// TIA Portal V20 export
FUNCTION_BLOCK "Side_Hydraulic"   // FB4, LAD
{ S7_Optimized_Access := 'TRUE' }
// stored: MemoryReserve 100, SetENOAutomatically false
   VAR_INPUT
      setUp : Bool;
      setDown : Bool;
      manual_Up : Bool;
      manual_Down : Bool;
      Sensor1_Up : Bool;
      Sensor1_Down : Bool;
      Sensor2_Up : Bool;
      Sensor2_Down : Bool;
      Reset : Bool;
   END_VAR
   VAR_OUTPUT
      Actuator_Up : Bool;
      Actuator_Down : Bool;
      Hydraulic_Unit : Bool;
      Alarm_Push_Actuators : Bool;
      Alarm_Pull_Actuators : Bool;
      Sensors_Down : Bool;
      Sensors_Up : Bool;
      Error : Bool;
   END_VAR
   VAR
      Time_to_PUSH_actuator { ExternalAccessible := 'False'; ExternalVisible := 'False'; ExternalWritable := 'False'} : TON_TIME;
      Time_to_PULL_actuator { S7_SetPoint := 'True'} : TON_TIME;
      Hydraulic_Unit_Timer { S7_SetPoint := 'True'} : TOF_TIME;
      TIMER_Pallet_UP { S7_SetPoint := 'True'} : TOF_TIME;
      TIMER_Pallet_DOWN { S7_SetPoint := 'True'} : TOF_TIME;
      Timer_Error { S7_SetPoint := 'True'} : TON_TIME;
      command_UP { ExternalAccessible := 'False'; ExternalVisible := 'False'; ExternalWritable := 'False'} : Bool;
      command_Down { ExternalAccessible := 'False'; ExternalVisible := 'False'; ExternalWritable := 'False'} : Bool;
   END_VAR
BEGIN

REGION Network 1: Sensors DOWN
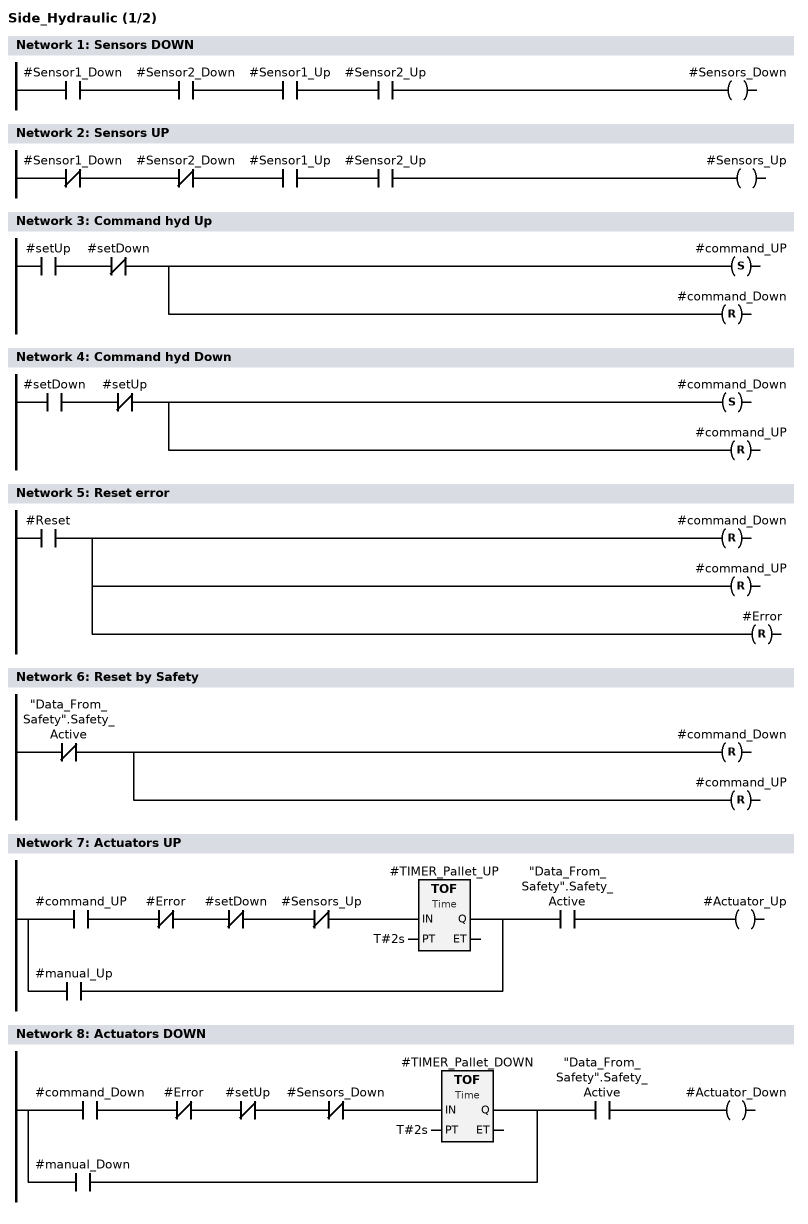
   RUNG wire#powerrail
      Contact( #Sensor1_Down )
      Contact( #Sensor2_Down )
      Contact( #Sensor1_Up )
      Contact( #Sensor2_Up )
      Coil( #Sensors_Down )
   END_RUNG
   // the same network as SCL:
   #Sensors_Down := #Sensor1_Down AND #Sensor2_Down AND #Sensor1_Up AND #Sensor2_Up;
END_REGION

REGION Network 2: Sensors UP
   RUNG wire#powerrail
      I_Contact( #Sensor1_Down )
      I_Contact( #Sensor2_Down )
      Contact( #Sensor1_Up )
      Contact( #Sensor2_Up )
      Coil( #Sensors_Up )
   END_RUNG
   // the same network as SCL:
   #Sensors_Up := NOT #Sensor1_Down AND NOT #Sensor2_Down AND #Sensor1_Up AND #Sensor2_Up;
END_REGION

REGION Network 3: Command hyd Up
   RUNG wire#powerrail
      Contact( #setUp )
      I_Contact( #setDown )
      wire#w1
      S_Coil( #command_UP )
   END_RUNG
   RUNG wire#w1
      R_Coil( #command_Down )
   END_RUNG
   // the same network as SCL:
   IF #setUp AND NOT #setDown THEN
       #command_UP := TRUE;
       #command_Down := FALSE;
   END_IF;
END_REGION

REGION Network 4: Command hyd Down
   RUNG wire#powerrail
      Contact( #setDown )
      I_Contact( #setUp )
      wire#w1
      S_Coil( #command_Down )
   END_RUNG
   RUNG wire#w1
      R_Coil( #command_UP )
   END_RUNG
   // the same network as SCL:
   IF #setDown AND NOT #setUp THEN
       #command_Down := TRUE;
       #command_UP := FALSE;
   END_IF;
END_REGION

REGION Network 5: Reset error
   RUNG wire#powerrail
      Contact( #Reset )
      wire#w1
      R_Coil( #command_Down )
   END_RUNG
   RUNG wire#w1
      R_Coil( #command_UP )
   END_RUNG
   RUNG wire#w1
      R_Coil( #Error )
   END_RUNG
   // the same network as SCL:
   IF #Reset THEN
       #command_Down := FALSE;
       #command_UP := FALSE;
       #Error := FALSE;
   END_IF;
END_REGION

REGION Network 6: Reset by Safety
   RUNG wire#powerrail
      I_Contact( "Data_From_Safety".Safety_Active )
      wire#w1
      R_Coil( #command_Down )
   END_RUNG
   RUNG wire#w1
      R_Coil( #command_UP )
   END_RUNG
   // the same network as SCL:
   IF NOT "Data_From_Safety".Safety_Active THEN
       #command_Down := FALSE;
       #command_UP := FALSE;
   END_IF;
END_REGION

REGION Network 7: Actuators UP
   RUNG wire#powerrail
      Contact( #command_UP )
      I_Contact( #Error )
      I_Contact( #setDown )
      I_Contact( #Sensors_Up )
      { S7_Templates := "time_type := Time" } #TIMER_Pallet_UP.TOF(pt := T#2s, et =>)
      wire#w1
      Contact( "Data_From_Safety".Safety_Active )
      Coil( #Actuator_Up )
   END_RUNG
   RUNG wire#powerrail
      Contact( #manual_Up )
   END_RUNG wire#w1
   // the same network as SCL:
   #TIMER_Pallet_UP(IN := #command_UP AND NOT #Error AND NOT #setDown AND NOT #Sensors_Up, PT := T#2s);   // TOF
   #Actuator_Up := (#TIMER_Pallet_UP.Q OR #manual_Up) AND "Data_From_Safety".Safety_Active;
END_REGION

REGION Network 8: Actuators DOWN
   RUNG wire#powerrail
      Contact( #command_Down )
      I_Contact( #Error )
      I_Contact( #setUp )
      I_Contact( #Sensors_Down )
      { S7_Templates := "time_type := Time" } #TIMER_Pallet_DOWN.TOF(pt := T#2s, et =>)
      wire#w1
      Contact( "Data_From_Safety".Safety_Active )
      Coil( #Actuator_Down )
   END_RUNG
   RUNG wire#powerrail
      Contact( #manual_Down )
   END_RUNG wire#w1
   // the same network as SCL:
   #TIMER_Pallet_DOWN(IN := #command_Down AND NOT #Error AND NOT #setUp AND NOT #Sensors_Down, PT := T#2s);   // TOF
   #Actuator_Down := (#TIMER_Pallet_DOWN.Q OR #manual_Down) AND "Data_From_Safety".Safety_Active;
END_REGION

REGION Network 9: Turn ON/OFF hydraulic unit
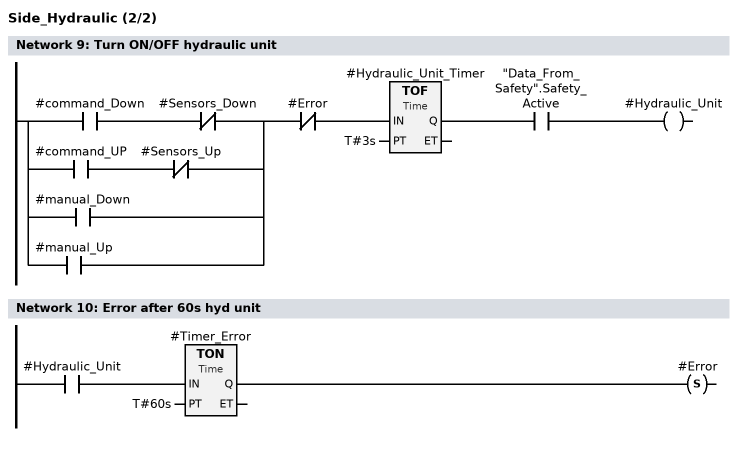
   RUNG wire#powerrail
      Contact( #command_Down )
      I_Contact( #Sensors_Down )
      wire#w1
      I_Contact( #Error )
      { S7_Templates := "time_type := Time" } #Hydraulic_Unit_Timer.TOF(pt := T#3s, et =>)
      Contact( "Data_From_Safety".Safety_Active )
      Coil( #Hydraulic_Unit )
   END_RUNG
   RUNG wire#powerrail
      Contact( #command_UP )
      I_Contact( #Sensors_Up )
   END_RUNG wire#w1
   RUNG wire#powerrail
      Contact( #manual_Down )
   END_RUNG wire#w1
   RUNG wire#powerrail
      Contact( #manual_Up )
   END_RUNG wire#w1
   // the same network as SCL:
   #Hydraulic_Unit_Timer(IN := ((#command_Down AND NOT #Sensors_Down) OR (#command_UP AND NOT #Sensors_Up) OR #manual_Down OR #manual_Up) AND NOT #Error,   // TOF
                         PT := T#3s);
   #Hydraulic_Unit := #Hydraulic_Unit_Timer.Q AND "Data_From_Safety".Safety_Active;
END_REGION

REGION Network 10: Error after 60s hyd unit
   RUNG wire#powerrail
      Contact( #Hydraulic_Unit )
      { S7_Templates := "time_type := Time" } #Timer_Error.TON(pt := T#60s, et =>)
      S_Coil( #Error )
   END_RUNG
   // the same network as SCL:
   #Timer_Error(IN := #Hydraulic_Unit, PT := T#60s);   // TON
   IF #Timer_Error.Q THEN #Error := TRUE; END_IF;
END_REGION
END_FUNCTION_BLOCK
